Fanuc KAREL source: compact_preamble.KL

PROGRAM KT00450
%NOLOCKGROUP
VAR
Y1 : ARRAY[2] OF BYTE
H2 : ARRAY[2] OF SHORT
OUT:BOOLEAN
BEGIN
Y1[1]=2
H2[1]=3
OUT=(Y1[1] >=H2[1])
END KT00450
